PROGRAM PRG_SFLX_02_OutfeedConvCtrl
VAR
	rsTransferNotConfirmed	: RS;
	rsOuterAtChuteExitNotConfirmed	: RS;

	tofOutfeedConvDelay	: FB_TOFR;
	rsExitRejectCtrl		: RS;

END_VAR

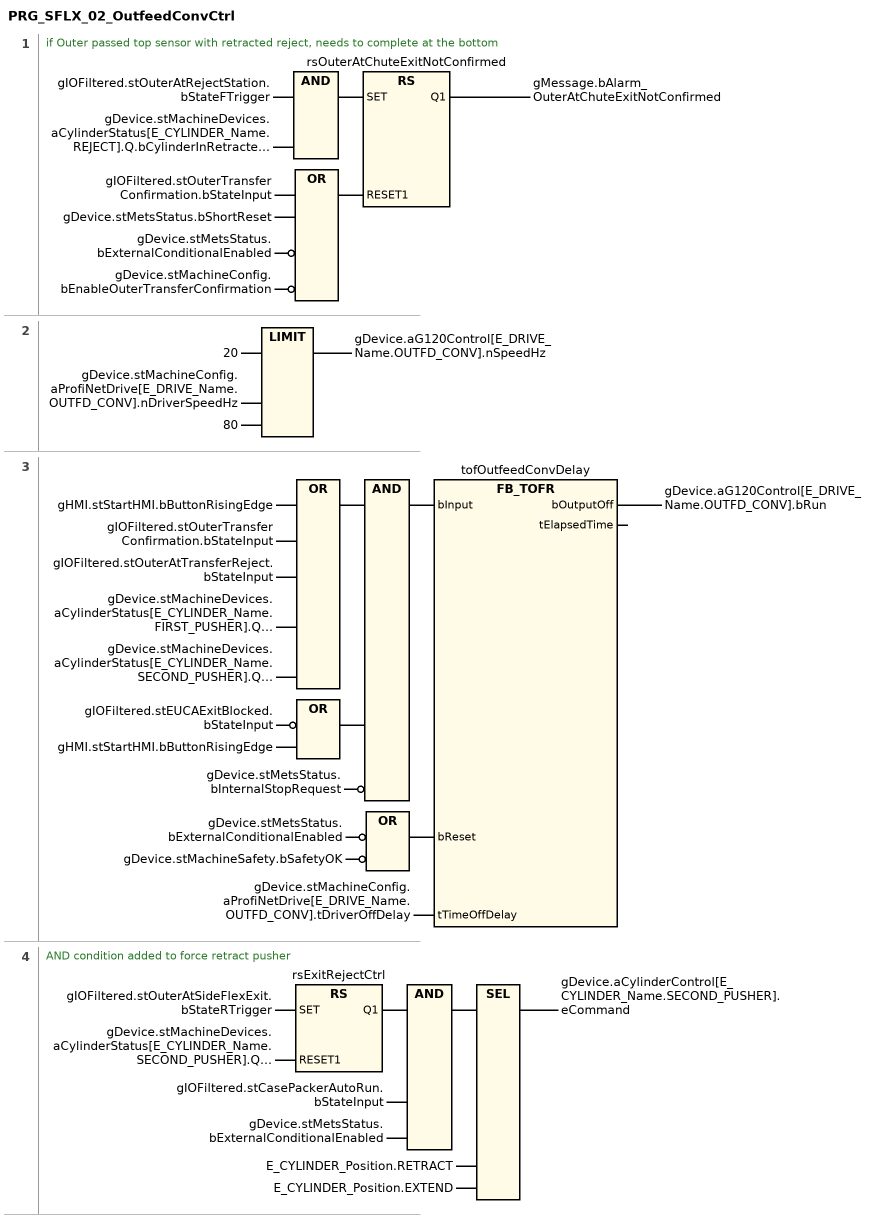
// NETWORK 1
// if Outer passed top sensor with retracted reject, needs to complete at the bottom
rsOuterAtChuteExitNotConfirmed(SET := gIOFiltered.stOuterAtRejectStation.bStateFTrigger AND gDevice.stMachineDevices.aCylinderStatus[E_CYLINDER_Name.REJECT].Q.bCylinderInRetractedPosition, RESET1 := gIOFiltered.stOuterTransferConfirmation.bStateInput OR gDevice.stMetsStatus.bShortReset OR NOT gDevice.stMetsStatus.bExternalConditionalEnabled OR NOT gDevice.stMachineConfig.bEnableOuterTransferConfirmation); // RS
gMessage.bAlarm_OuterAtChuteExitNotConfirmed := rsOuterAtChuteExitNotConfirmed.Q1;

// NETWORK 2
gDevice.aG120Control[E_DRIVE_Name.OUTFD_CONV].nSpeedHz := LIMIT(20, gDevice.stMachineConfig.aProfiNetDrive[E_DRIVE_Name.OUTFD_CONV].nDriverSpeedHz, 80);

// NETWORK 3
tofOutfeedConvDelay(
    bInput := (gHMI.stStartHMI.bButtonRisingEdge OR gIOFiltered.stOuterTransferConfirmation.bStateInput OR gIOFiltered.stOuterAtTransferReject.bStateInput OR gDevice.stMachineDevices.aCylinderStatus[E_CYLINDER_Name.FIRST_PUSHER].Q.bCylinderIsExtending OR gDevice.stMachineDevices.aCylinderStatus[E_CYLINDER_Name.SECOND_PUSHER].Q.bCylinderIsRetracting) AND (NOT gIOFiltered.stEUCAExitBlocked.bStateInput OR gHMI.stStartHMI.bButtonRisingEdge) AND NOT gDevice.stMetsStatus.bInternalStopRequest,
    bReset := NOT gDevice.stMetsStatus.bExternalConditionalEnabled OR NOT gDevice.stMachineSafety.bSafetyOK,
    tTimeOffDelay := gDevice.stMachineConfig.aProfiNetDrive[E_DRIVE_Name.OUTFD_CONV].tDriverOffDelay); // FB_TOFR
gDevice.aG120Control[E_DRIVE_Name.OUTFD_CONV].bRun := tofOutfeedConvDelay.bOutputOff;

// NETWORK 4
// AND condition added to force retract pusher
rsExitRejectCtrl(SET := gIOFiltered.stOuterAtSideFlexExit.bStateRTrigger, RESET1 := gDevice.stMachineDevices.aCylinderStatus[E_CYLINDER_Name.SECOND_PUSHER].Q.bCylinderInExtendedPosition); // RS
gDevice.aCylinderControl[E_CYLINDER_Name.SECOND_PUSHER].eCommand := SEL(rsExitRejectCtrl.Q1 AND gIOFiltered.stCasePackerAutoRun.bStateInput AND gDevice.stMetsStatus.bExternalConditionalEnabled, E_CYLINDER_Position.RETRACT, E_CYLINDER_Position.EXTEND);

END_PROGRAM

(* stored: Version 1.1.0.1
   POU PRG_SFLX_02_OutfeedConvCtrl: Id {81b7f9d2-39f8-4f0b-8362-81c1b1fe750d}, SpecialFunc None *)
